// TwinCAT 3 PLC project TcSpeech_Sample
// ProgramVersion: 3.1.4026.9
// libraries:
//   Tc2_Standard, * (Beckhoff Automation GmbH)
//   Tc2_System, * (Beckhoff Automation GmbH)
//   Tc3_Speech, * (Beckhoff Automation GmbH)
// project tree:
//   / PlcTask.TcTTO
//   POUs/ MAIN.TcPOU, MainASR.TcPOU, MainTTS.TcPOU
// real-time tasks:
//   TASK PlcTask: cycle T#10ms, priority 20, ADS port 350

CONFIGURATION TcSpeech_Sample
    RESOURCE PLC ON TwinCAT3
        TASK PlcTask(INTERVAL := T#10ms, PRIORITY := 20);
        PROGRAM MAIN WITH PlcTask : MAIN;
    END_RESOURCE
END_CONFIGURATION

// ---- POUs/MAIN.TcPOU
// TwinCAT Speech Sample for Speech Recognition and Text-To-Speech (simple)
// This example shows only the most necessary code.
// Start Recognition or Start Text-To-Speech can be triggered in respective PRGs
// MainASR: PRG for Speech Recognition
// MainTTS: PRG for Text-To-Speech
PROGRAM MAIN

MainTTS();
MainASR();

END_PROGRAM

// ---- POUs/MainTTS.TcPOU
// Text-To-Speech can be triggered by setting bSpeak to true
// Configured languages are 1033 (English (United States), default) and 1031 (German) --> "nLanguageId" variable to switch
PROGRAM MainTTS
VAR
// TTS Variables
bSpeak			    : BOOL 			:= FALSE;
{attribute 'TcEncoding':= 'UTF-8'}
sText2Speech        : STRING(4095)  := '<speak>TcSpeech demo project is greeting you.</speak>';


// TTS Configuration
nConfigIdTTS	: UINT 				:= 200;
nLanguageId     : UINT 				:= 1033;
fbTTS 			: FB_TextToSpeech 	:= (nConfigurationId := nConfigIdTTS, nLanguageId := nLanguageId); 

END_VAR

// Set bSpeak to true, to start a speech synthesis
IF bSpeak THEN 
	fbTTS(sUtterance := sText2Speech, bSpeak := TRUE, nConfigurationId:= nConfigIdTTS);
	
	IF NOT fbTTS.bBusy THEN
		fbTTS(sUtterance := sText2Speech,bSpeak := FALSE, nConfigurationId:= nConfigIdTTS);
		bSpeak := FALSE;
	END_IF
END_IF

END_PROGRAM

// ---- POUs/MainASR.TcPOU
// Start Recognition can be triggered by setting bListen to true
// "Hello TwinCAT" is configured to be recognized
// If recognition is detected, variable bRecognition is set to true for 1 second
PROGRAM MainASR
VAR 
// Start speech recognition by setting to true
bListen			: BOOL 	:= FALSE;

// If "Hello TwinCAT" is recognized bRecognition is set to true for 1 sec
bRecognition	: BOOL;

// ASR Configuration
nConfigIdASR    : UINT 					:= 100;
fbASR 			: FB_SpeechRecognition	:= (nConfigurationId := nConfigIdASR);

// ASR Variables                               
nLastRecoId    	: ULINT 				:= 0;

timer	: TON;
END_VAR

// Set bListen to true, to start speech recognition
fbASR(bListen := bListen, nConfigurationId:= nConfigIdASR);

// If new recognition is available and recognition confidence is high enough (over 70%) set bRecognition to true
IF nLastRecoId <> fbASR.nRecognitionId THEN
	nLastRecoId := fbASR.nRecognitionId;
	IF fbAsr.fRecognitionConfidence > 0.7 THEN
	  bRecognition := TRUE;
	END_IF
END_IF


// Keep bRecognition true for just a second
IF bRecognition THEN
	timer(IN := TRUE, PT := T#1S);
	IF timer.Q THEN
		timer(IN := FALSE);
		bRecognition := FALSE;
	END_IF
END_IF

END_PROGRAM
